TYPE OutputBase_10CEE7DE :
STRUCT
END_STRUCT
END_TYPE

(* stored: Version 1.2.0.0, ProductVersion 3.1.4024.9
   DUT OutputBase_10CEE7DE: Id {78535f8a-bc2e-4e32-9d31-2d8282c18a58} *)
